Staubli VAL3: getPathInstr.pgx

public program getPathInstr(string x_sInstr (dimensions=1), string& x_sPath (dimensions=1))
begin
  // give back the path of the Instruction
  if isDefined(iInstruction[x_sInstr])
    x_sPath=iInstruction[x_sInstr].sPath
  else
    x_sPath=""
  endIf
end
